PROGRAM MAIN
VAR
	fbCoalDrill 	: FB_Drill ; 
	fbcopperDrill	: FB_Drill ;
	fbIronDrill		: FB_Drill ;
	test : int;
		
	iCoalStash 		: UINT ; // total amount of coal
	iCopperOreStash : UINT ; // total amount of copper stored
	iIronOreStash	: UINT ; // Total amount of iron ore stash  
	
	fbIronProduction_1 		: FB_StoneFurnace;
	fbCopperProduction_1	: FB_StoneFurnace;
	
END_VAR


CollectOre();
ProduceIron();
CollectCopperOre();
test:=1;

METHOD CollectCopperOre : BOOL
VAR_INPUT
END_VAR
	fbCopperProduction_1();
END_METHOD

METHOD CollectOre : BOOL
VAR_INPUT
END_VAR
// run Drills
	fbCoalDrill(); 
	fbcopperDrill();
	fbIronDrill();

// collect ore
	iCoalStash 		:= iCoalStash + fbCoalDrill.ProductsOut;
	iCopperOreStash := iCopperOreStash + fbcopperDrill.ProductsOut;
	iIronOreStash	:= iIronOreStash + fbIronDrill.ProductsOut;
END_METHOD

METHOD ProduceIron : BOOL
VAR_INPUT
END_VAR

// run production
	fbIronProduction_1();
END_METHOD

END_PROGRAM

(* stored: Version 1.1.0.1, ProductVersion 3.1.4026.8
   POU MAIN: Id {9779ac30-3bb2-408e-a339-e7064e52c5d5}, SpecialFunc None
   Method CollectCopperOre: Id {926e8480-a214-43ab-89e0-27855abfcb55}
   Method CollectOre: Id {7a33b17c-4198-4c6d-b1f2-b13e3198d9b9}
   Method ProduceIron: Id {c24eebcd-2226-43d2-9b45-29968881bd3b} *)
